Yaskawa INFORM job: L_F_TOP_1_S1.JBI

/JOB
//NAME L_F_TOP_1_S1
//POS
///NPOS 16,16,16,0,0,0
///TOOL 2
///POSTYPE PULSE
///PULSE
C00000=-124128,-6471,-18196,-31354,22369,47411
C00001=-123392,11873,-48916,-48580,43474,56574
C00002=-122848,18417,-47199,-50932,44894,57492
C00003=-122638,21058,-46436,-51897,45421,57865
C00004=-125315,38031,-27819,-40802,29487,39996
C00005=-125279,37918,-27917,-40880,29727,39099
C00006=-125889,-3007,-63124,-42237,31473,39970
C00007=-125400,23376,-44119,-32479,18960,19891
C00008=-126023,52865,-25571,-31587,3254,10086
C00009=-118500,43294,-23330,-35343,371,7589
C00010=-117573,42357,-22816,-35801,31,7259
C00011=-118605,43340,-23300,-38079,-719,8343
C00012=-119634,44543,-23752,-40253,-1568,9437
C00013=-120162,46074,-21562,-40008,-2199,9345
C00014=-121429,50037,-15922,-39455,-3804,9105
C00015=-121872,34193,12974,-45374,-22188,1903
///TOOL 0
BC00000=104847
BC00001=104847
BC00002=104847
BC00003=104847
BC00004=104847
BC00005=104847
BC00006=104847
BC00007=104847
BC00008=104847
BC00009=104847
BC00010=104847
BC00011=104847
BC00012=104847
BC00013=104847
BC00014=104847
BC00015=104847
EC00000=-184118,1883
EC00001=-184118,1883
EC00002=-184118,1883
EC00003=-184118,1883
EC00004=-184118,1883
EC00005=-184118,1883
EC00006=-184118,1883
EC00007=-184118,1883
EC00008=-184118,1883
EC00009=-184118,1883
EC00010=-184118,1883
EC00011=-184118,1883
EC00012=-184118,1883
EC00013=-184118,1883
EC00014=-184118,1883
EC00015=-184118,1883
//INST
///DATE 2026/05/13 10:02
///ATTR SC,RW
///GROUP1 RB1,BS1
///GROUP2 ST1
NOP
'L_F_top_1_s1
MEMOF
CLEAR MPF
'Path W1
SSFTOF
MOVJ C00000 BC00000 VJ=100.00  +MOVJ EC00000 VJ=100.00
SMOVL C00001 BC00001 V=1000.0  +MOVJ EC00001
SMOVL C00002 BC00002 V=400.0  +MOVJ EC00002
SMOVL C00003 BC00003 V=10.0 PL=0  +MOVJ EC00003
SMOVL C00004 BC00004 V=10.0  +MOVJ EC00004
SMOVL C00005 BC00005 V=10.0  +MOVJ EC00005
SMOVL C00006 BC00006 V=10.0  +MOVJ EC00006
SMOVL C00007 BC00007 V=10.0  +MOVJ EC00007
SMOVL C00008 BC00008 V=10.0  +MOVJ EC00008
SMOVL C00009 BC00009 V=10.0  +MOVJ EC00009
SMOVL C00010 BC00010 V=10.0  +MOVJ EC00010
SMOVL C00011 BC00011 V=10.0  +MOVJ EC00011
SMOVL C00012 BC00012 V=10.0  +MOVJ EC00012
SMOVL C00013 BC00013 V=400.0  +MOVJ EC00013
SMOVL C00014 BC00014 V=1000.0  +MOVJ EC00014
SMOVL C00015 BC00015 V=1000.0  +MOVJ EC00015
'EndPath W1
END
